{attribute 'Tc2GvlVarNames'}
VAR_GLOBAL
	fbConcat		: FB_CONCAT;
    fbSystemTime	: FB_SystemTimeService;
END_VAR

(* stored: Version 1.1.0.1, ProductVersion 3.1.4026.18
   GVL GVL_GLOBAL: Id {3bae080b-6d51-42a6-ac5f-9ecf21d00dbf} *)
